(* Logix 5000 project; controller cal1615 1756-L62 rev 20.11; software revision 20.05; part 57 of 82 *)
(* tags used below, declared in another part *)
   FAULT : BOOL;   // Fault AFI
   HMI : BOOL;   // AFI HMI
   p01r09_pb_global_reset : BOOL;   // System Modes PB: Global Fault Reset
   p02_dint_to_hmi : hmi_dint;   // MOP HMI Iface Dint to HMI
   p24_do_edge_guide_input_1 : BOOL;   // Edge Guide Digital Output Input 1
   p24r01 : routine;
   p24r04 : routine;   // Edge Control Outputs
   p24r04_timer_fault : TIMER[4];   // Edge Control Outputs Fault Delay
   p24r04_timer_warning : TIMER[4];   // Edge Control Outputs Warning Dwell
   p24r05 : routine;   // Edge Control Dint to HMI
   p24r05_timer_fault : TIMER[4];   // Edge Control Dint to HMI Fault Dwell
   p24r05_timer_warning : TIMER[4];   // Edge Control Dint to HMI Warning Delay
   p24r06 : routine;   // Edge Control Real to HMI
   p24r06_timer_fault : TIMER[4];   // Edge Control Real to HMI Fault Delay
   p24r06_timer_warning : TIMER[4];   // Edge Control Real to HMI Warning Delay
   p24r07 : routine;   // Edge Control Alarms
   p24r07_timer_fault : TIMER[4];   // Edge Control Alarms Fault Delay
   p24r07_timer_warning : TIMER[4];   // Edge Control Alarms Warning Delay
   p24r08 : routine;   // Edge Control Warings
   p24r08_timer_fault : TIMER[4];   // Edge Control Warnings Fault Delay
   p24r08_timer_warning : TIMER[4];   // Edge Control Warnings Warning Delay
   p24r09 : routine;   // Tension Stand 2 Modes
   p24r09_timer_fault : TIMER[4];   // Edge Control Modes Fault Delay
   p24r09_timer_warning : TIMER[4];   // Edge Control Modes Warning Delay
(* P24_Edge_Control, continued *)

ROUTINE R04_Outputs   (* ladder *)
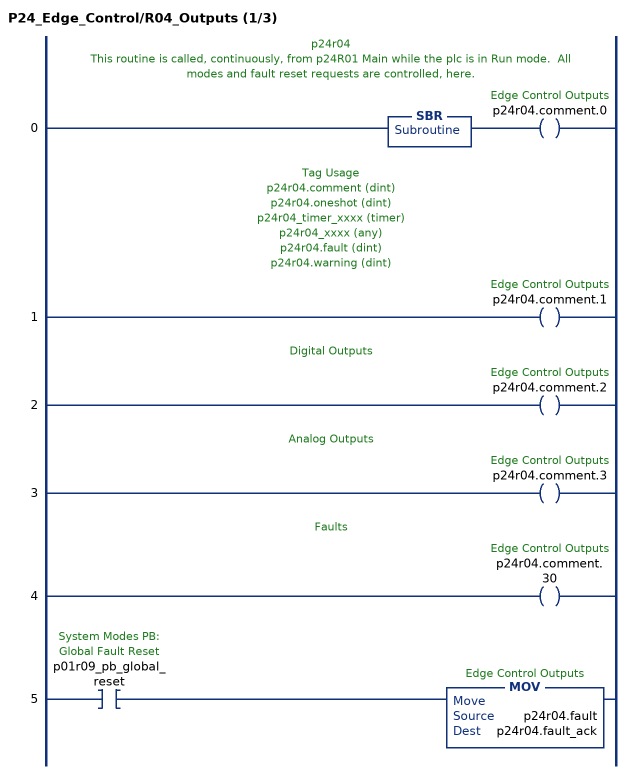
   // p24r04
   // This routine is called, continuously, from p24R01 Main while the plc is in Run mode.  All modes and fault reset requests are controlled, here.
   0: SBR()OTE(p24r04.comment.0);
   // Tag Usage
   // p24r04.comment (dint)
   // p24r04.oneshot (dint)
   // p24r04_timer_xxxx (timer)
   // p24r04_xxxx (any)
   // p24r04.fault (dint)
   // p24r04.warning (dint)
   1: OTE(p24r04.comment.1);
   // Digital Outputs
   2: OTE(p24r04.comment.2);
   // Analog Outputs
   3: OTE(p24r04.comment.3);
   // Faults
   4: OTE(p24r04.comment.30);
   5: XIC(p01r09_pb_global_reset)MOV(p24r04.fault,p24r04.fault_ack);
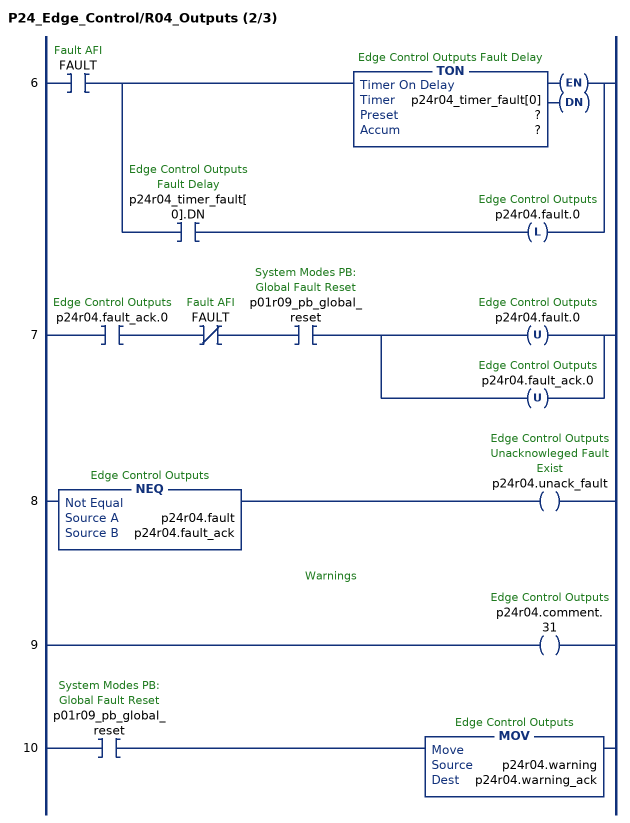
   6: XIC(FAULT)[TON(p24r04_timer_fault[0],?,?) ,XIC(p24r04_timer_fault[0].DN) OTL(p24r04.fault.0) ];
   7: XIC(p24r04.fault_ack.0)XIO(FAULT)XIC(p01r09_pb_global_reset)[OTU(p24r04.fault.0) ,OTU(p24r04.fault_ack.0) ];
   8: NEQ(p24r04.fault,p24r04.fault_ack)OTE(p24r04.unack_fault);
   // Warnings
   9: OTE(p24r04.comment.31);
   10: XIC(p01r09_pb_global_reset)MOV(p24r04.warning,p24r04.warning_ack);
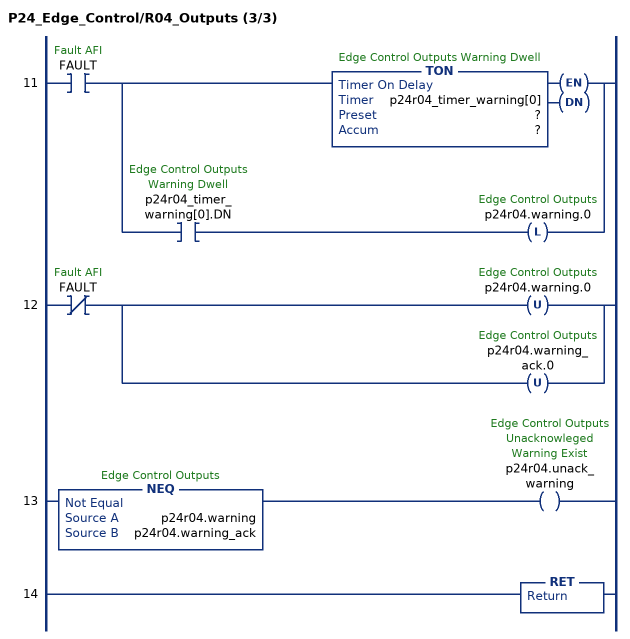
   11: XIC(FAULT)[TON(p24r04_timer_warning[0],?,?) ,XIC(p24r04_timer_warning[0].DN) OTL(p24r04.warning.0) ];
   12: XIO(FAULT)[OTU(p24r04.warning.0) ,OTU(p24r04.warning_ack.0) ];
   13: NEQ(p24r04.warning,p24r04.warning_ack)OTE(p24r04.unack_warning);
   14: RET();
END_ROUTINE

ROUTINE R05_Dint_to_HMI   (* ladder *)
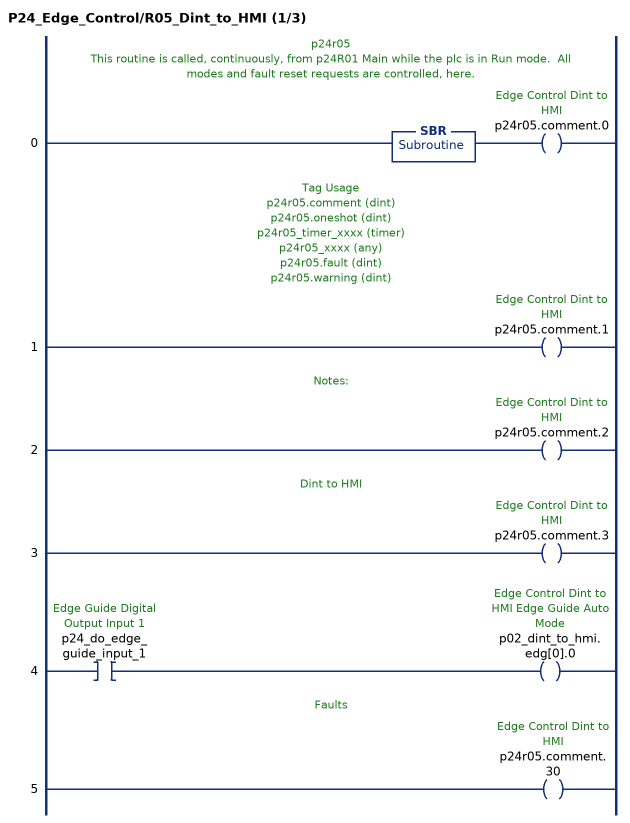
   // p24r05
   // This routine is called, continuously, from p24R01 Main while the plc is in Run mode.  All modes and fault reset requests are controlled, here.
   0: SBR()OTE(p24r05.comment.0);
   // Tag Usage
   // p24r05.comment (dint)
   // p24r05.oneshot (dint)
   // p24r05_timer_xxxx (timer)
   // p24r05_xxxx (any)
   // p24r05.fault (dint)
   // p24r05.warning (dint)
   1: OTE(p24r05.comment.1);
   // Notes:
   2: OTE(p24r05.comment.2);
   // Dint to HMI
   3: OTE(p24r05.comment.3);
   4: XIC(p24_do_edge_guide_input_1)OTE(p02_dint_to_hmi.edg[0].0);
   // Faults
   5: OTE(p24r05.comment.30);
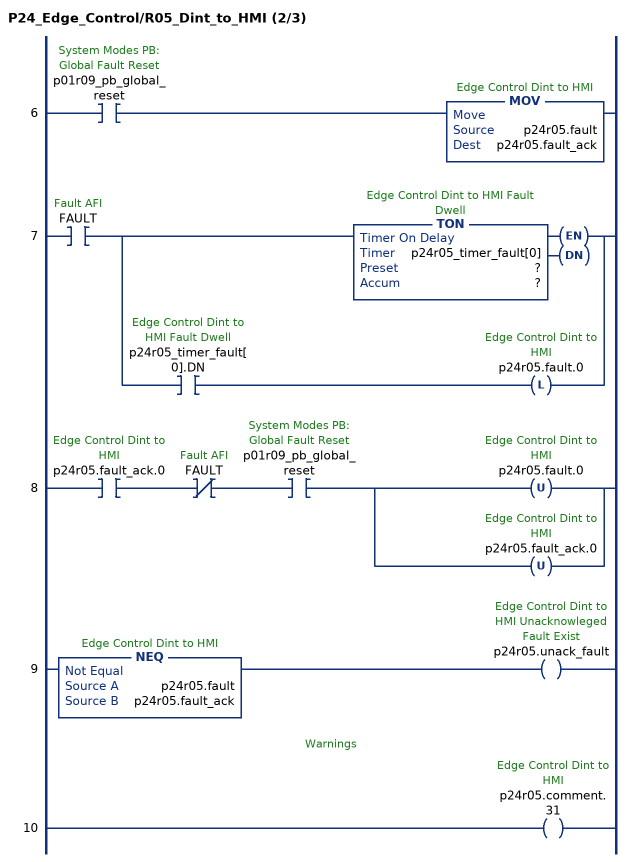
   6: XIC(p01r09_pb_global_reset)MOV(p24r05.fault,p24r05.fault_ack);
   7: XIC(FAULT)[TON(p24r05_timer_fault[0],?,?) ,XIC(p24r05_timer_fault[0].DN) OTL(p24r05.fault.0) ];
   8: XIC(p24r05.fault_ack.0)XIO(FAULT)XIC(p01r09_pb_global_reset)[OTU(p24r05.fault.0) ,OTU(p24r05.fault_ack.0) ];
   9: NEQ(p24r05.fault,p24r05.fault_ack)OTE(p24r05.unack_fault);
   // Warnings
   10: OTE(p24r05.comment.31);
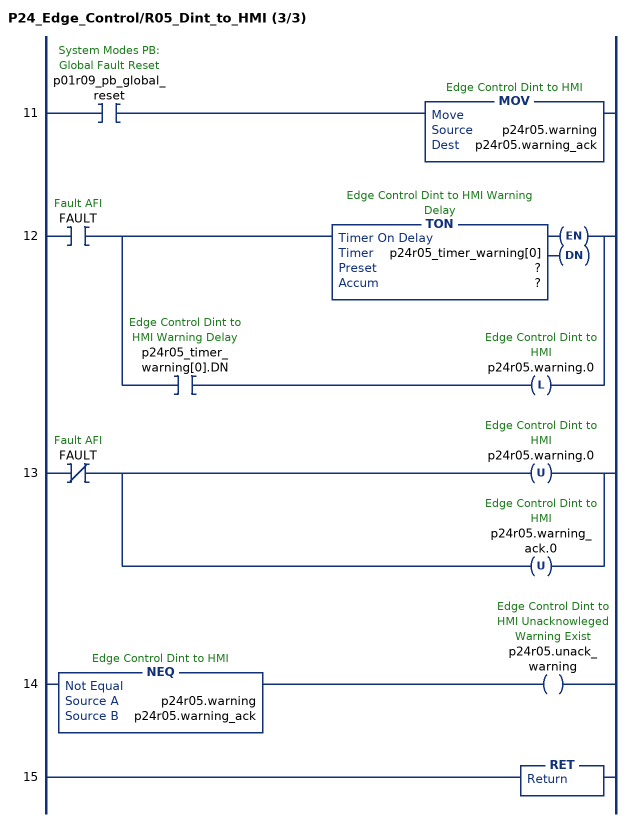
   11: XIC(p01r09_pb_global_reset)MOV(p24r05.warning,p24r05.warning_ack);
   12: XIC(FAULT)[TON(p24r05_timer_warning[0],?,?) ,XIC(p24r05_timer_warning[0].DN) OTL(p24r05.warning.0) ];
   13: XIO(FAULT)[OTU(p24r05.warning.0) ,OTU(p24r05.warning_ack.0) ];
   14: NEQ(p24r05.warning,p24r05.warning_ack)OTE(p24r05.unack_warning);
   15: RET();
END_ROUTINE

ROUTINE R06_Real_to_HMI   (* ladder *)
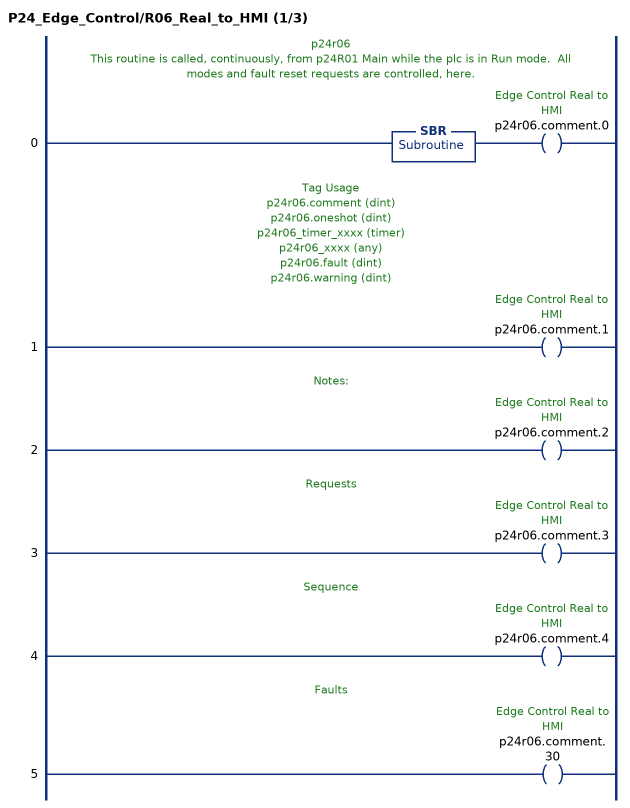
   // p24r06
   // This routine is called, continuously, from p24R01 Main while the plc is in Run mode.  All modes and fault reset requests are controlled, here.
   0: SBR()OTE(p24r06.comment.0);
   // Tag Usage
   // p24r06.comment (dint)
   // p24r06.oneshot (dint)
   // p24r06_timer_xxxx (timer)
   // p24r06_xxxx (any)
   // p24r06.fault (dint)
   // p24r06.warning (dint)
   1: OTE(p24r06.comment.1);
   // Notes:
   2: OTE(p24r06.comment.2);
   // Requests
   3: OTE(p24r06.comment.3);
   // Sequence
   4: OTE(p24r06.comment.4);
   // Faults
   5: OTE(p24r06.comment.30);
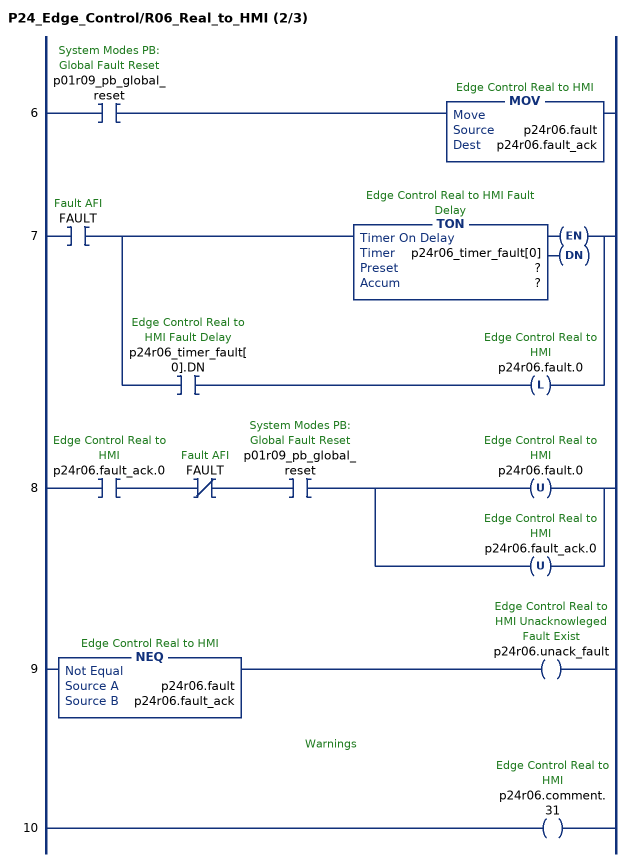
   6: XIC(p01r09_pb_global_reset)MOV(p24r06.fault,p24r06.fault_ack);
   7: XIC(FAULT)[TON(p24r06_timer_fault[0],?,?) ,XIC(p24r06_timer_fault[0].DN) OTL(p24r06.fault.0) ];
   8: XIC(p24r06.fault_ack.0)XIO(FAULT)XIC(p01r09_pb_global_reset)[OTU(p24r06.fault.0) ,OTU(p24r06.fault_ack.0) ];
   9: NEQ(p24r06.fault,p24r06.fault_ack)OTE(p24r06.unack_fault);
   // Warnings
   10: OTE(p24r06.comment.31);
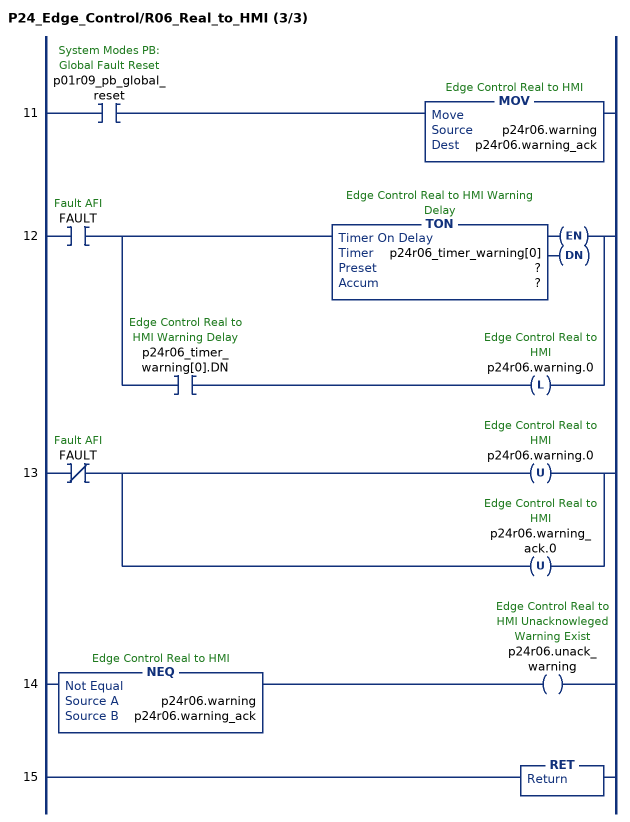
   11: XIC(p01r09_pb_global_reset)MOV(p24r06.warning,p24r06.warning_ack);
   12: XIC(FAULT)[TON(p24r06_timer_warning[0],?,?) ,XIC(p24r06_timer_warning[0].DN) OTL(p24r06.warning.0) ];
   13: XIO(FAULT)[OTU(p24r06.warning.0) ,OTU(p24r06.warning_ack.0) ];
   14: NEQ(p24r06.warning,p24r06.warning_ack)OTE(p24r06.unack_warning);
   15: RET();
END_ROUTINE

ROUTINE R07_Alarms   (* ladder *)
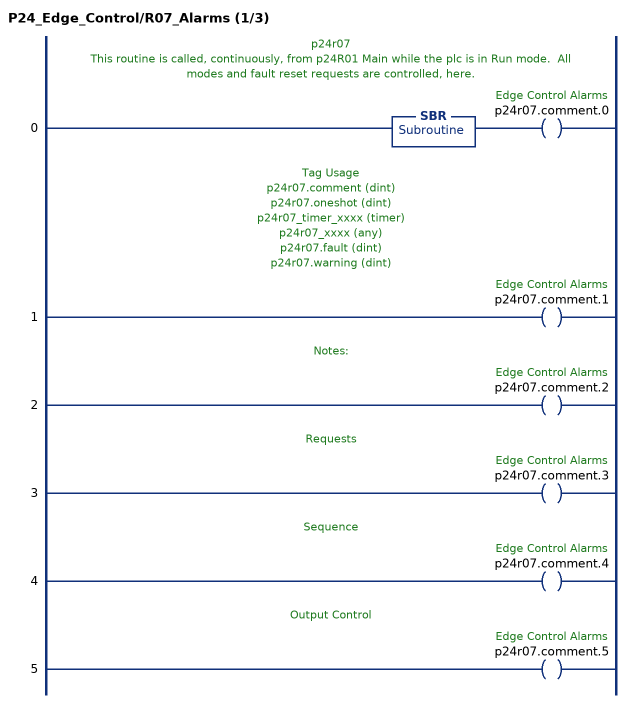
   // p24r07
   // This routine is called, continuously, from p24R01 Main while the plc is in Run mode.  All modes and fault reset requests are controlled, here.
   0: SBR()OTE(p24r07.comment.0);
   // Tag Usage
   // p24r07.comment (dint)
   // p24r07.oneshot (dint)
   // p24r07_timer_xxxx (timer)
   // p24r07_xxxx (any)
   // p24r07.fault (dint)
   // p24r07.warning (dint)
   1: OTE(p24r07.comment.1);
   // Notes:
   2: OTE(p24r07.comment.2);
   // Requests
   3: OTE(p24r07.comment.3);
   // Sequence
   4: OTE(p24r07.comment.4);
   // Output Control
   5: OTE(p24r07.comment.5);
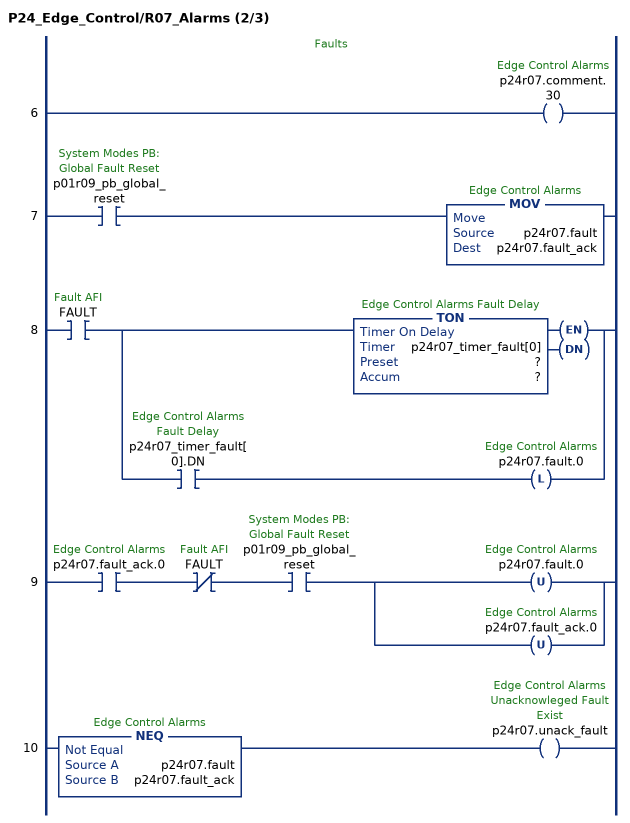
   // Faults
   6: OTE(p24r07.comment.30);
   7: XIC(p01r09_pb_global_reset)MOV(p24r07.fault,p24r07.fault_ack);
   8: XIC(FAULT)[TON(p24r07_timer_fault[0],?,?) ,XIC(p24r07_timer_fault[0].DN) OTL(p24r07.fault.0) ];
   9: XIC(p24r07.fault_ack.0)XIO(FAULT)XIC(p01r09_pb_global_reset)[OTU(p24r07.fault.0) ,OTU(p24r07.fault_ack.0) ];
   10: NEQ(p24r07.fault,p24r07.fault_ack)OTE(p24r07.unack_fault);
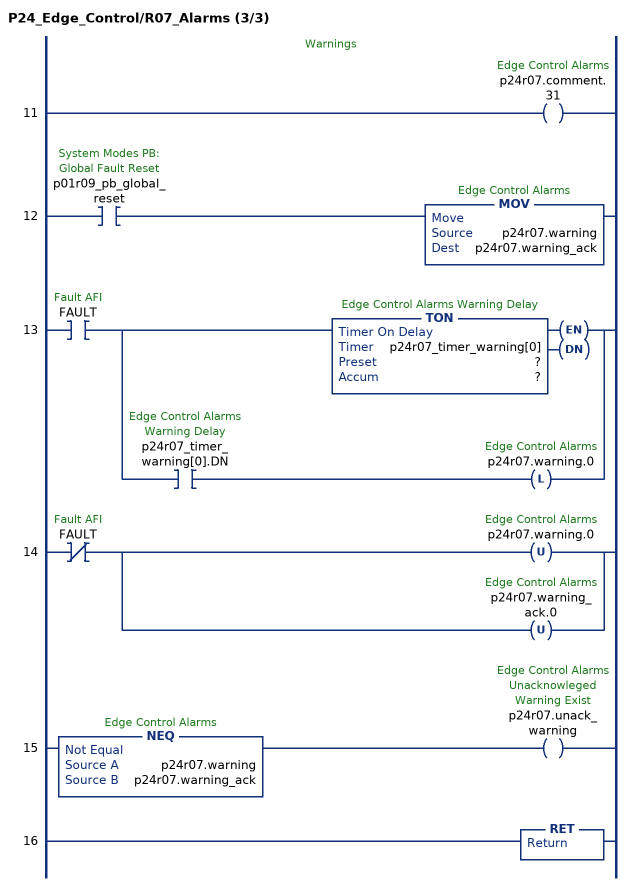
   // Warnings
   11: OTE(p24r07.comment.31);
   12: XIC(p01r09_pb_global_reset)MOV(p24r07.warning,p24r07.warning_ack);
   13: XIC(FAULT)[TON(p24r07_timer_warning[0],?,?) ,XIC(p24r07_timer_warning[0].DN) OTL(p24r07.warning.0) ];
   14: XIO(FAULT)[OTU(p24r07.warning.0) ,OTU(p24r07.warning_ack.0) ];
   15: NEQ(p24r07.warning,p24r07.warning_ack)OTE(p24r07.unack_warning);
   16: RET();
END_ROUTINE

ROUTINE R08_Warnings   (* ladder *)
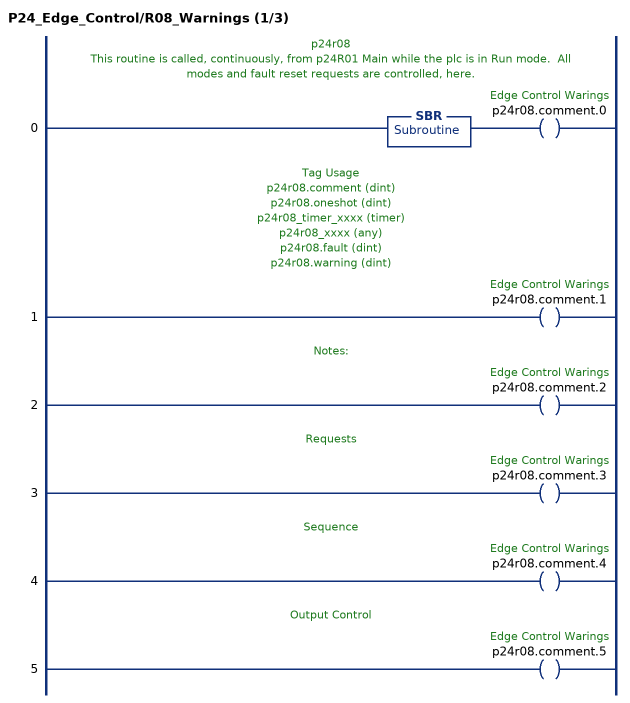
   // p24r08
   // This routine is called, continuously, from p24R01 Main while the plc is in Run mode.  All modes and fault reset requests are controlled, here.
   0: SBR()OTE(p24r08.comment.0);
   // Tag Usage
   // p24r08.comment (dint)
   // p24r08.oneshot (dint)
   // p24r08_timer_xxxx (timer)
   // p24r08_xxxx (any)
   // p24r08.fault (dint)
   // p24r08.warning (dint)
   1: OTE(p24r08.comment.1);
   // Notes:
   2: OTE(p24r08.comment.2);
   // Requests
   3: OTE(p24r08.comment.3);
   // Sequence
   4: OTE(p24r08.comment.4);
   // Output Control
   5: OTE(p24r08.comment.5);
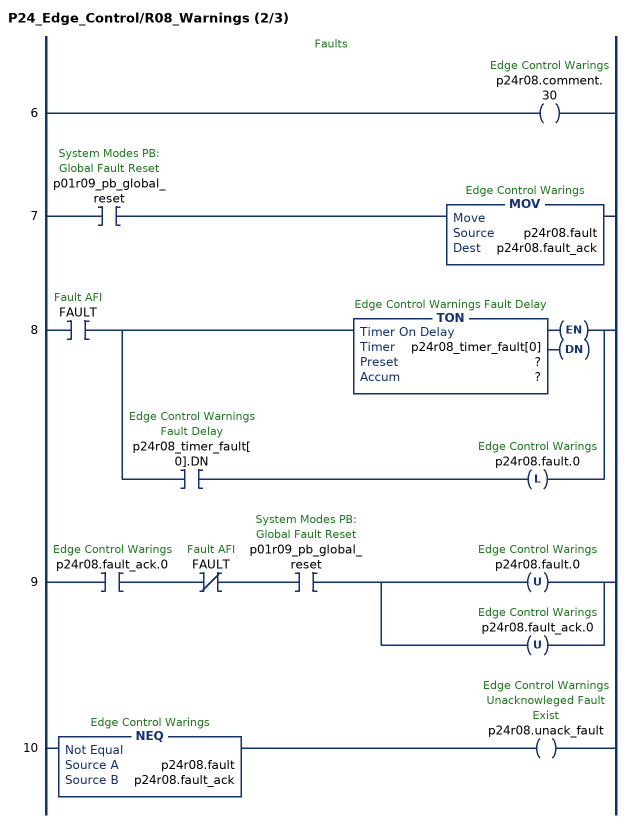
   // Faults
   6: OTE(p24r08.comment.30);
   7: XIC(p01r09_pb_global_reset)MOV(p24r08.fault,p24r08.fault_ack);
   8: XIC(FAULT)[TON(p24r08_timer_fault[0],?,?) ,XIC(p24r08_timer_fault[0].DN) OTL(p24r08.fault.0) ];
   9: XIC(p24r08.fault_ack.0)XIO(FAULT)XIC(p01r09_pb_global_reset)[OTU(p24r08.fault.0) ,OTU(p24r08.fault_ack.0) ];
   10: NEQ(p24r08.fault,p24r08.fault_ack)OTE(p24r08.unack_fault);
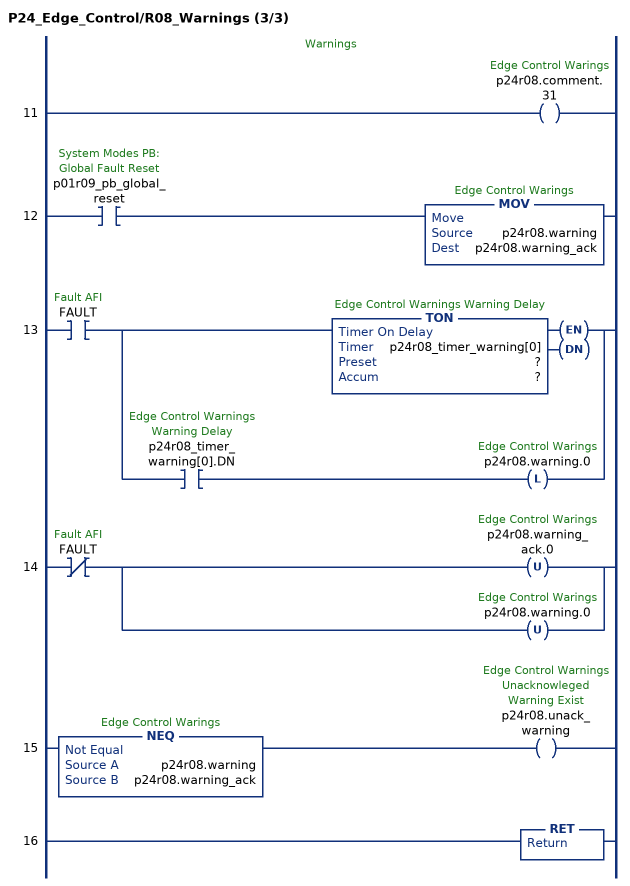
   // Warnings
   11: OTE(p24r08.comment.31);
   12: XIC(p01r09_pb_global_reset)MOV(p24r08.warning,p24r08.warning_ack);
   13: XIC(FAULT)[TON(p24r08_timer_warning[0],?,?) ,XIC(p24r08_timer_warning[0].DN) OTL(p24r08.warning.0) ];
   14: XIO(FAULT)[OTU(p24r08.warning_ack.0) ,OTU(p24r08.warning.0) ];
   15: NEQ(p24r08.warning,p24r08.warning_ack)OTE(p24r08.unack_warning);
   16: RET();
END_ROUTINE

ROUTINE R09_Modes   (* ladder *)
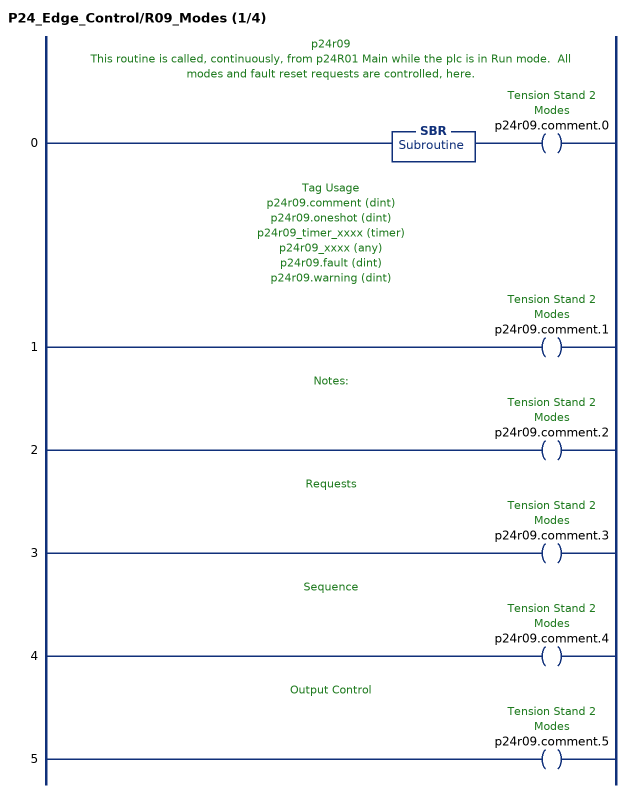
   // p24r09
   // This routine is called, continuously, from p24R01 Main while the plc is in Run mode.  All modes and fault reset requests are controlled, here.
   0: SBR()OTE(p24r09.comment.0);
   // Tag Usage
   // p24r09.comment (dint)
   // p24r09.oneshot (dint)
   // p24r09_timer_xxxx (timer)
   // p24r09_xxxx (any)
   // p24r09.fault (dint)
   // p24r09.warning (dint)
   1: OTE(p24r09.comment.1);
   // Notes:
   2: OTE(p24r09.comment.2);
   // Requests
   3: OTE(p24r09.comment.3);
   // Sequence
   4: OTE(p24r09.comment.4);
   // Output Control
   5: OTE(p24r09.comment.5);
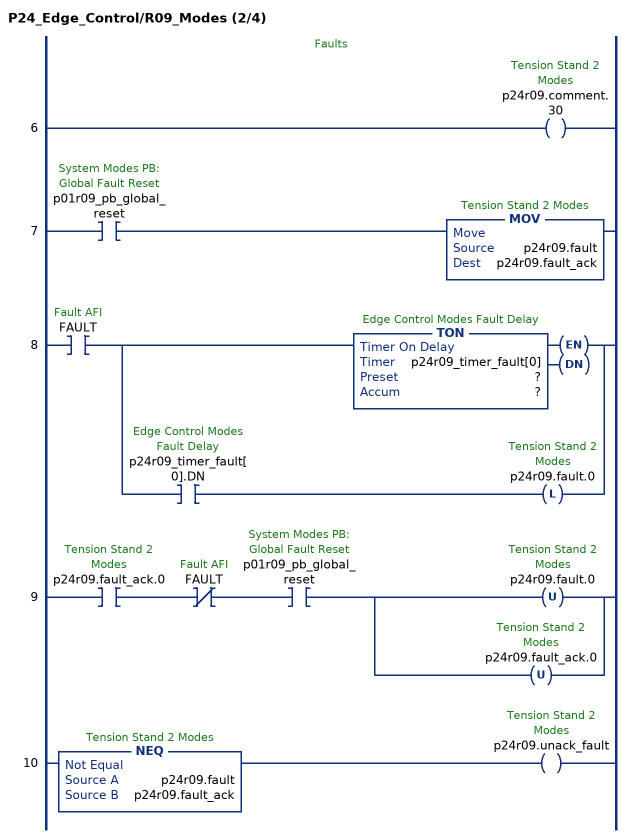
   // Faults
   6: OTE(p24r09.comment.30);
   7: XIC(p01r09_pb_global_reset)MOV(p24r09.fault,p24r09.fault_ack);
   8: XIC(FAULT)[TON(p24r09_timer_fault[0],?,?) ,XIC(p24r09_timer_fault[0].DN) OTL(p24r09.fault.0) ];
   9: XIC(p24r09.fault_ack.0)XIO(FAULT)XIC(p01r09_pb_global_reset)[OTU(p24r09.fault.0) ,OTU(p24r09.fault_ack.0) ];
   10: NEQ(p24r09.fault,p24r09.fault_ack)OTE(p24r09.unack_fault);
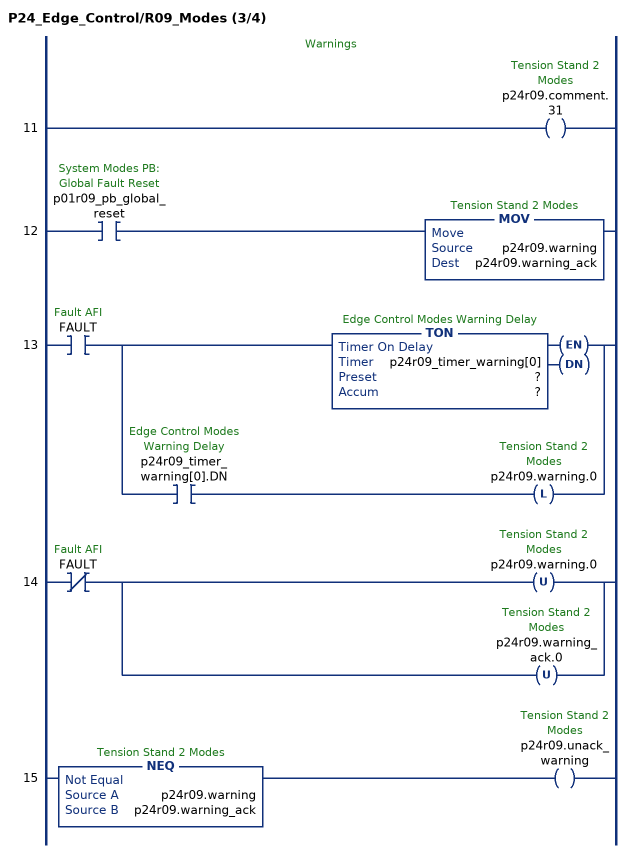
   // Warnings
   11: OTE(p24r09.comment.31);
   12: XIC(p01r09_pb_global_reset)MOV(p24r09.warning,p24r09.warning_ack);
   13: XIC(FAULT)[TON(p24r09_timer_warning[0],?,?) ,XIC(p24r09_timer_warning[0].DN) OTL(p24r09.warning.0) ];
   14: XIO(FAULT)[OTU(p24r09.warning.0) ,OTU(p24r09.warning_ack.0) ];
   15: NEQ(p24r09.warning,p24r09.warning_ack)OTE(p24r09.unack_warning);
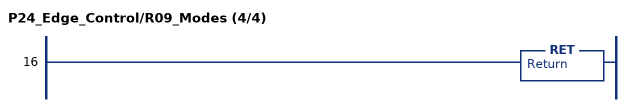
   16: RET();
END_ROUTINE
